(* PLC project ifmCR711S_TemplateProject, CODESYS CODESYS V3.5 SP11 *)
(* stored: creationDateTime 2026-08-04T14:35:54.4941509, version 2.4.10.0, modificationDateTime 2026-08-04T14:25:20.5601505, organization ifm electronic *)
(* Project template with CR711S configured 2.25MByte Standard 2.25MByte Safety *)

PROGRAM FB_TESTING
  VAR CONSTANT
    uiMinVoltage : UINT := 5000;  (* Minimum Voltage in mV *)
  END_VAR
  VAR
    fbSystemSupply : ifmIOcommon.SystemSupply;  (* Function Block to monitor supply voltage on VBB15 (from ignition) *)
    fbSupplySwitch : ifmIOcommon.SupplySwitch;  (* Function Block to turn ON/OFF latching switch on VBB15 supply (from ignition) *)
    uiCurrSupplyVolt : UINT;  (* Operating Voltage in mV *)
    TOF_0 : TOF;
  END_VAR

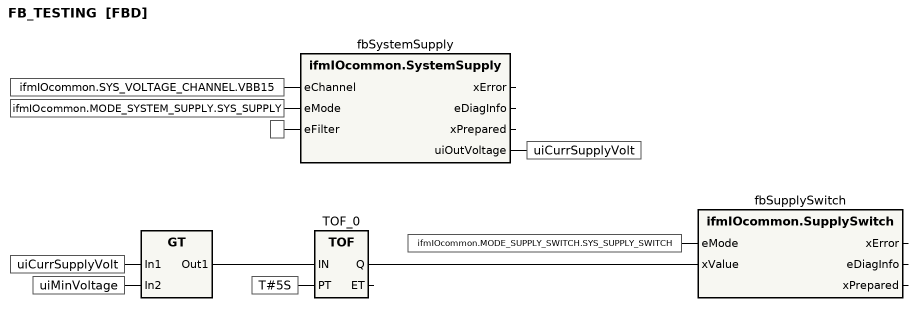
(* FBD diagram, written out as Structured Text *)
(* // Function Block to monitor supply voltage on VBB15 (from ignition) *)
fbSystemSupply(eChannel := ifmIOcommon.SYS_VOLTAGE_CHANNEL.VBB15, eMode := ifmIOcommon.MODE_SYSTEM_SUPPLY.SYS_SUPPLY, eFilter := , uiOutVoltage => uiCurrSupplyVolt);
(* //Safely power off PLC when ignition (VBB15) is lower than 5V for more than 10s. Enable timer on falling edge *)
TOF_0(IN := uiCurrSupplyVolt > uiMinVoltage, PT := T#5S);
fbSupplySwitch(eMode := ifmIOcommon.MODE_SUPPLY_SWITCH.SYS_SUPPLY_SWITCH, xValue := TOF_0.Q);
END_PROGRAM
